FUNCTION_BLOCK DataDemux
  (* Version 1.0, 2007-08-28, Goran Cengic, Chalmers *)
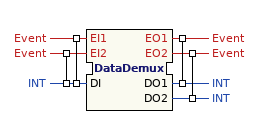
  EVENT_INPUT
    EI1 WITH DI;
    EI2 WITH DI;
  END_EVENT
  EVENT_OUTPUT
    EO1 WITH DO1;
    EO2 WITH DO2;
  END_EVENT
  VAR_INPUT
    DI : INT;
  END_VAR
  VAR_OUTPUT
    DO1 : INT;
    DO2 : INT;
  END_VAR
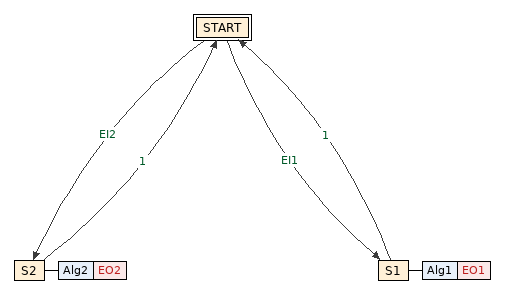
  EC_STATES
    START;
    S1 : Alg1 -> EO1;
    S2 : Alg2 -> EO2;
  END_STATES
  EC_TRANSITIONS
    START TO S1 := EI1;
    S1 TO START := 1;
    START TO S2 := EI2;
    S2 TO START := 1;
  END_TRANSITIONS
  ALGORITHM Alg1 IN Java:
DO1 = DI;
  END_ALGORITHM
  ALGORITHM Alg2 IN Java:
DO2 = DI;
  END_ALGORITHM
END_FUNCTION_BLOCK
